FUNCTION_BLOCK E_REND
  (* Version 1.0, 2005-11-20, Goran Cengic, Chalmers *)
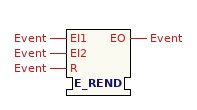
  EVENT_INPUT
    EI1;
    EI2;
    R;
  END_EVENT
  EVENT_OUTPUT
    EO;
  END_EVENT
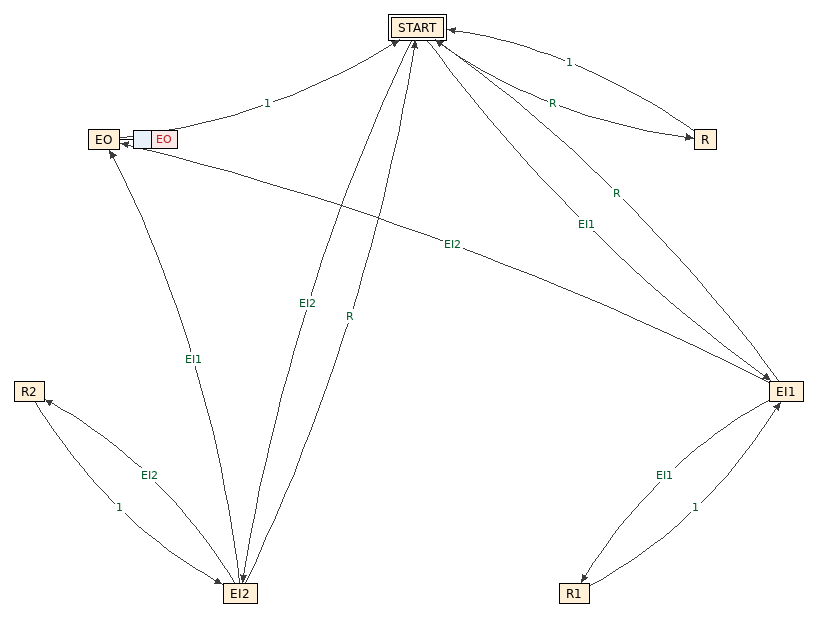
  EC_STATES
    START;
    R;
    EI1;
    R1;
    EI2;
    R2;
    EO : -> EO;
  END_STATES
  EC_TRANSITIONS
    START TO R := R;
    R TO START := 1;
    START TO EI1 := EI1;
    EI1 TO START := R;
    START TO EI2 := EI2;
    EI2 TO START := R;
    EI1 TO R1 := EI1;
    R1 TO EI1 := 1;
    EI1 TO EO := EI2;
    EI2 TO R2 := EI2;
    R2 TO EI2 := 1;
    EI2 TO EO := EI1;
    EO TO START := 1;
  END_TRANSITIONS
END_FUNCTION_BLOCK
